(* PLC project Simulator, SUTD Blank 1.0 *)
(* stored: creationDateTime 2016-05-18T21:14:07, modificationDateTime 2020-03-10T00:36:37, language en-US *)

PROGRAM Stage1
  VAR
    LIT101 AT %IW1 : REAL;  (* Stage 1 Water Level [Input] *)
    MV101 AT %QX1.0 : BOOL;  (* Water tank Input Pump [Output] *)
    P101 AT %QX1.1 : BOOL;  (* Water tank Output Pump [Output] *)
  END_VAR
  VAR CONSTANT
    HIGH_LIMIT : REAL := 800.0;  (* High water level threshold *)
    LOW_LIMIT : REAL := 500.0;  (* Low water level threshold *)
  END_VAR

            
IF LIT101 > HIGH_LIMIT THEN
  MV101:=0;
  P101:=1;
ELSIF LIT101 < LOW_LIMIT THEN
  MV101:=1;
  P101:=0;
END_IF;
          
END_PROGRAM

CONFIGURATION Config0
  RESOURCE Res0 ON PLC
    TASK TaskMain(INTERVAL := T#5ms, PRIORITY := 0);
    PROGRAM Inst0 WITH TaskMain : Stage1;
  END_RESOURCE
END_CONFIGURATION
